(* LS Electric XG5000 project: Study4_Counter *)
(* PLC LSPLC *)
(* module base 0 slot 0: 입력 모듈:XGI-D21A (DC 24V 입력, 8점 (전류소스/싱크입력)) *)
(* module base 0 slot 1: 출력 모듈:XGQ-RY1A (릴레이 출력, 8점 (2A용, 단독 COM.)) *)

PROGRAM NewProgram (* task: 스캔 프로그램 *)
VAR
    다운카운터 : CTD_INT;
    다운카운터1 : CTD_INT;
    리셋 : BOOL;
    스위치 AT %IX0.0.0 : BOOL;
    스위치2 AT %IX0.0.1 : BOOL;
    양변환검출코일 : BOOL;
    양변환스위치 : BOOL;
    업다운카운터 : CTUD_INT;
    업카운터1 : CTU_INT;
    업카운터2 : CTU_INT;
    카운트다운시작 : BOOL := 0;
END_VAR

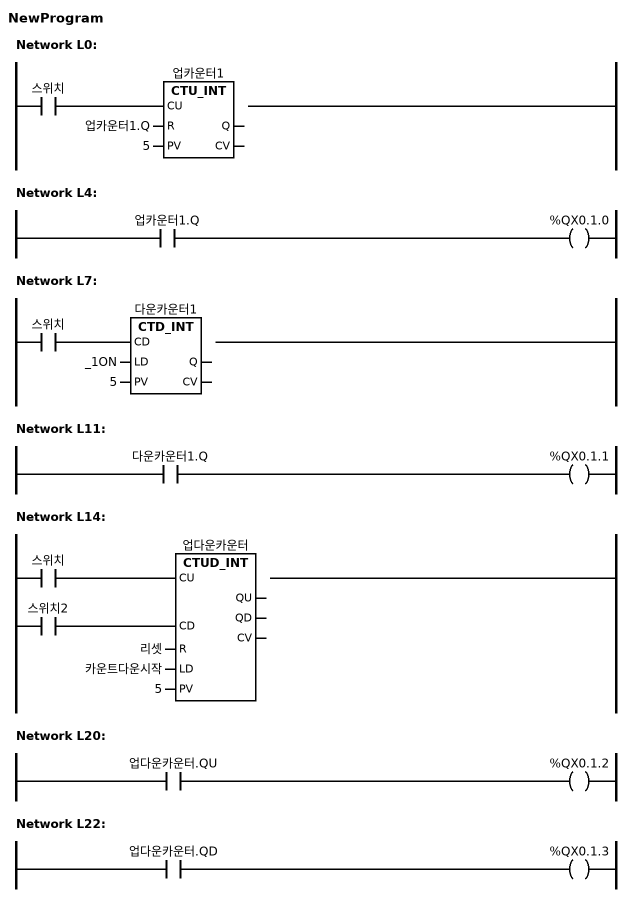
(* Rung L0 *)
업카운터1(CU := 스위치, R := 업카운터1.Q, PV := 5);
(* Rung L4 *)
%QX0.1.0 := 업카운터1.Q;
(* Rung L7 *)
다운카운터1(CD := 스위치, LD := _1ON, PV := 5);
(* Rung L11 *)
%QX0.1.1 := 다운카운터1.Q;
(* Rung L14 *)
업다운카운터(CU := 스위치, CD := 스위치2, R := 리셋, LD := 카운트다운시작, PV := 5);
(* Rung L20 *)
%QX0.1.2 := 업다운카운터.QU;
(* Rung L22 *)
%QX0.1.3 := 업다운카운터.QD;
END_PROGRAM